{attribute 'GeneratedUsingTerminal: EL5102-0000-0016'}
{attribute addProperty BoxType "EL5102-0000-0016"}
{attribute addProperty Id "Enable_latch_CBOOL1Enable_latch_extern_on_positive_edgeBOOL1Set_counterBOOL1Enable_latch_extern_on_negative_edgeBOOL1Set_counter_on_latch_CBOOL1Set_software_gateBOOL1Set_counter_on_latch_extern_on_positive_edgeBOOL1Set_counter_on_latch_extern_on_negative_edgeBOOL1Enable_latch_extern_2_on_positive_edgeBOOL1Enable_latch_extern_2_on_negative_edgeBOOL1"}
{attribute addProperty CRC "3572750464"}
{attribute addProperty Size "10"}
TYPE Control_D4F3D880 :
STRUCT
	{attribute addProperty Name "Enable_latch_C"}
	Enable_latch_C : BOOL;
	{attribute addProperty Name "Enable_latch_extern_on_positive_edge"}
	Enable_latch_extern_on_positive_edge : BOOL;
	{attribute addProperty Name "Set_counter"}
	Set_counter : BOOL;
	{attribute addProperty Name "Enable_latch_extern_on_negative_edge"}
	Enable_latch_extern_on_negative_edge : BOOL;
	{attribute addProperty Name "Set_counter_on_latch_C"}
	Set_counter_on_latch_C : BOOL;
	{attribute addProperty Name "Set_software_gate"}
	Set_software_gate : BOOL;
	{attribute addProperty Name "Set_counter_on_latch_extern_on_positive_edge"}
	Set_counter_on_latch_extern_on_positive_edge : BOOL;
	{attribute addProperty Name "Set_counter_on_latch_extern_on_negative_edge"}
	Set_counter_on_latch_extern_on_negative_edge : BOOL;
	{attribute addProperty Name "Enable_latch_extern_2_on_positive_edge"}
	Enable_latch_extern_2_on_positive_edge : BOOL;
	{attribute addProperty Name "Enable_latch_extern_2_on_negative_edge"}
	Enable_latch_extern_2_on_negative_edge : BOOL;
END_STRUCT
END_TYPE

(* stored: Version 1.2.0.0, ProductVersion 3.1.4024.9
   DUT Control_D4F3D880: Id {32ae0c1a-b191-4e32-b4a5-e0f0dd7cf0d1} *)
